TYPE structHBMSerialCtrl :
STRUCT
	In_Init:BOOL;
	In_Trigger:BOOL;
	
	Out_ReceiveDone:BOOL;
	Out_WeightResult:REAL;
	Out_InitOK:BOOL;	
	Out_ErrorWord:INT;
	Out_ErrorString:STRING;

END_STRUCT
END_TYPE

(* stored: Version 1.1.0.1, ProductVersion 3.1.4018.2
   DUT structHBMSerialCtrl: Id {c14d29c4-1683-4d46-839f-d799045b6a54} *)
